FUNCTION F_TimeFromString : LINT
VAR_INPUT
	sTime : STRING(31);
END_VAR

F_TimeFromString :=  ULINT_TO_LINT(DCTIME64_TO_FILETIME64(STRING_TO_DCTIME64(sTime)));

END_FUNCTION

(* stored: Version 1.1.0.1
   POU F_TimeFromString: Id {d84117b3-d38d-4228-b42e-ab885218d446}, SpecialFunc None *)
